// TwinCAT 3 PLC project MAXI
// ProgramVersion: 3.1.4024.0
// libraries:
//   Tc2_Standard, * (Beckhoff Automation GmbH)
//   Tc2_System, * (Beckhoff Automation GmbH)
//   Tc2_Utilities, * (Beckhoff Automation GmbH)
//   Tc3_Module, * (Beckhoff Automation GmbH)
// project tree:
//   DUTs/ BufferState.TcDUT
//   GVLs/ globals.TcGVL (not stored)
//   / PlcTask.TcTTO
//   POUs/ AnalogInput.TcPOU, FemtoCtrl.TcPOU, FilterRingBuffer.TcPOU (not stored), FlowMeter.TcPOU, LED.TcPOU, MAIN.TcPOU, ValueBuffer.TcPOU
// real-time tasks:
//   TASK PlcTask: cycle T#1ms, priority 20, ADS port 350
// I/O:
//   DEVICE Device 1 (EtherCAT), AmsNetId 5.82.117.74.2.1
//     Term 1 (EK1200) [EK1200-5000 EtherCAT Power supply (2A E-Bus)]
//       Term 2 (EL2595) [EL2595 1Ch. LED constant current terminal]
//       Term 3 (EL2595) [EL2595 1Ch. LED constant current terminal]
//       Term 4 (EL3102) [EL3102 2Ch. Ana. Input +/-10V, Diff.]
//       Term 5 (ELM3004-0000) [ELM3004-0000 4Ch. Ana. Input +/-30V, 24 bit, high precision]
//       Term 6 (EL9505) [EL9505 Power supply terminal 5V]
//       Term 7 (EL1124) [EL1124 4Ch. Dig. Input 5V, 10µs, Sensor Power]
//       Term 8 (EL2124) [EL2124 4Ch. Dig. Output 5V, 20mA]
//       Term 9 (EL2124) [EL2124 4Ch. Dig. Output 5V, 20mA]
//       Term 10 (EL2124) [EL2124 4Ch. Dig. Output 5V, 20mA]
//       Term 11 (EL9011) [EL9011 End Terminal]
// variable links:
//   MAXI/MAXI Instance <-> Device 1 (EtherCAT)/Term 1 (EK1200)/Term 2 (EL2595)
//     PlcTask Inputs/MAIN.LedBlue.bOutputActive <-> DOX Status/Status/Output active
//     PlcTask Inputs/MAIN.LedBlue.nCurrent <-> DOX Synchron info data/Info data 2
//     PlcTask Outputs/MAIN.LedBlue.bOutputSetpoint <-> DOX Control/Control/Output
//   MAXI/MAXI Instance <-> Device 1 (EtherCAT)/Term 1 (EK1200)/Term 3 (EL2595)
//     PlcTask Inputs/MAIN.LedWhite.bOutputActive <-> DOX Status/Status/Output active
//     PlcTask Inputs/MAIN.LedWhite.nCurrent <-> DOX Synchron info data/Info data 2
//     PlcTask Outputs/MAIN.LedWhite.bOutputSetpoint <-> DOX Control/Control/Output
//   MAXI/MAXI Instance <-> Device 1 (EtherCAT)/Term 1 (EK1200)/Term 5 (ELM3004-0000)
//     PlcTask Inputs/MAIN.ADC{1..4}.nRawValue <-> PAI Samples 1 Channel {1..4}/Samples[0]  (4 links)
//   MAXI/MAXI Instance <-> Device 1 (EtherCAT)/Term 1 (EK1200)/Term 7 (EL1124)
//     PlcTask Inputs/MAIN.Femto1.bOverload <-> Channel 1/Input
//     PlcTask Inputs/MAIN.Femto2.bOverload <-> Channel 3/Input
//     PlcTask Inputs/MAIN.flowmeter.bReedSwitch <-> Channel 2/Input
//   MAXI/MAXI Instance <-> Device 1 (EtherCAT)/Term 1 (EK1200)/Term 8 (EL2124)
//     PlcTask Outputs/MAIN.Femto1.bGainMode <-> Channel 4/Output
//     PlcTask Outputs/MAIN.Femto1.nGainBits <-> Channel 1/Output
//     PlcTask Outputs/MAIN.Femto1.nGainBits @bit 1 <-> Channel 2/Output
//     PlcTask Outputs/MAIN.Femto1.nGainBits @bit 2 <-> Channel 3/Output
//   MAXI/MAXI Instance <-> Device 1 (EtherCAT)/Term 1 (EK1200)/Term 9 (EL2124)
//     PlcTask Outputs/MAIN.Femto2.bGainMode <-> Channel 4/Output
//     PlcTask Outputs/MAIN.Femto2.nGainBits <-> Channel 1/Output
//     PlcTask Outputs/MAIN.Femto2.nGainBits @bit 1 <-> Channel 2/Output
//     PlcTask Outputs/MAIN.Femto2.nGainBits @bit 2 <-> Channel 3/Output

CONFIGURATION MAXI
    RESOURCE PLC ON TwinCAT3
        TASK PlcTask(INTERVAL := T#1ms, PRIORITY := 20);
        PROGRAM MAIN WITH PlcTask : MAIN;
    END_RESOURCE
END_CONFIGURATION

// ---- DUTs/BufferState.TcDUT
{attribute 'qualified_only'}
{attribute 'strict'}
TYPE BufferState :
(
	INIT, IDLE, STORING, FULL
);
END_TYPE

// ---- POUs/MAIN.TcPOU
PROGRAM MAIN
VAR
	LedBlue: LED;
	LedWhite: LED;
	Femto1: FemtoCtrl;
	Femto2: FemtoCtrl;
	ADC1: AnalogInput;
	ADC2: AnalogInput;
	ADC3: AnalogInput;
	ADC4: AnalogInput;
	bStartBuffer: BOOL := TRUE;
	bPrepareBuffer: BOOL := FALSE;
	nAdcBufferSize: UDINT := 1000; // size of array for dedicated acquisitions 
	bStopAdcBuffer: BOOL := FALSE;
	flowmeter: FlowMeter;
	sCommand: STRING := '';
	bCommandExecute: BOOL := FALSE;
	sCommandResult: STRING := '';
	fb_Shutdown: NT_Shutdown;
END_VAR

LedBlue();
LedWhite();
ADC1();
ADC2();
ADC3();
ADC4();

flowmeter();

IF bPrepareBuffer THEN
	nAdcBufferSize := ADC1.valuebuffer.PrepareBuffer(nNumValues:=nAdcBufferSize);
	nAdcBufferSize := ADC2.valuebuffer.PrepareBuffer(nNumValues:=nAdcBufferSize);
	nAdcBufferSize := ADC3.valuebuffer.PrepareBuffer(nNumValues:=nAdcBufferSize);
	nAdcBufferSize := ADC4.valuebuffer.PrepareBuffer(nNumValues:=nAdcBufferSize);
	bPrepareBuffer := FALSE;
END_IF

IF bStopAdcBuffer THEN
	ADC1.valuebuffer.StopBuffer();
	ADC2.valuebuffer.StopBuffer();
	ADC3.valuebuffer.StopBuffer();
	ADC4.valuebuffer.StopBuffer();
	bStopAdcBuffer := FALSE;
END_IF

IF bStartBuffer THEN
	ADC1.valuebuffer.StartBuffer();
	ADC2.valuebuffer.StartBuffer();
	ADC3.valuebuffer.StartBuffer();
	ADC4.valuebuffer.StartBuffer();
	bStartBuffer := FALSE;
END_IF

IF bCommandExecute THEN
	IF sCommand = 'SHUTDOWN' THEN
		fb_Shutdown(NETID:='', DELAY:=0, START:=bCommandExecute);
		sCommandResult := 'shutting down';
	ELSE
		sCommandResult := 'unknown command';
	END_IF
	bCommandExecute := FALSE;
END_IF

END_PROGRAM

// ---- POUs/LED.TcPOU
FUNCTION_BLOCK LED
VAR
	bOutputActive AT %I*: BOOL;
	bOutputSetpoint AT %Q*: BOOL;
	nCurrent AT %I*: UINT;
	nOutputCurrent: UINT;
END_VAR

IF bOutputActive THEN
	nOutputCurrent := nCurrent;
ELSE
	nOutputCurrent := 0;
END_IF

END_FUNCTION_BLOCK

// ---- POUs/FemtoCtrl.TcPOU
FUNCTION_BLOCK FemtoCtrl
VAR
	nGainBits AT %Q*: WORD; // assign multiple output bits with correct offset
	bGainMode AT %Q*: BOOL := TRUE; // TRUE: low noise, FALSE: high speed
	bOverload AT %I*: BOOL;
END_VAR

METHOD GetGain : WORD
VAR_INPUT
END_VAR
GetGain := nGainBits;
END_METHOD

METHOD GetGainMode : BOOL
VAR_INPUT
END_VAR
GetGainMode := bGainMode;
END_METHOD

METHOD GetOverload : BOOL
VAR_INPUT
END_VAR
GetOverload := bOverload;
END_METHOD

METHOD SetGain
VAR_INPUT
	nGain: WORD;
END_VAR
nGainBits := nGain;
END_METHOD

METHOD SetGainMode
VAR_INPUT
	bGainHigh: BOOL;
END_VAR
bGainMode := bGainHigh;
END_METHOD

END_FUNCTION_BLOCK

// ---- POUs/AnalogInput.TcPOU
FUNCTION_BLOCK AnalogInput
VAR
	nMaxRawValue: REAL := 7812500;  // for 24 bit device, e.g. ELM300x - check manual
	nRawValue AT %I*: DINT; // signed 32 bit integer representing full value range
	fMaxVoltage: REAL := 10; // measurement range
	valuebuffer: ValueBuffer; // buffer for timed measurements
	filterbuffer: FilterRingBuffer;
	nFilterSize: UDINT := 100;
	fVoltage: REAL;
	fVoltageFiltered: REAL; // running average filter
END_VAR

fVoltage := fMaxVoltage * DINT_TO_REAL(nRawValue) / nMaxRawValue;  

IF filterbuffer.nBufferSize <> nFilterSize THEN
	nFilterSize := filterbuffer.SetFilterSize(nFilterSize);
END_IF
filterbuffer.Store(fVoltage);
fVoltageFiltered := filterbuffer.CalculateMean();

valuebuffer(fValue:=fVoltage);  // makes sure buffer in initialized and calls StoreValueConditional

END_FUNCTION_BLOCK

// ---- POUs/ValueBuffer.TcPOU
FUNCTION_BLOCK ValueBuffer
VAR_INPUT
	fValue : REAL;
END_VAR
VAR
	values: ARRAY[0 .. globals.MAX_BUFFER_LENGTH] OF REAL;
	bInitialized: BOOL:=FALSE;
	nStoreEveryNthValue : UINT:=1;
	nCurrentIndex : UDINT:=1;
	eBufState : BufferState:=BufferState.INIT;
	nBufSize : UDINT:=1000;
	nTickCount : UDINT;
END_VAR

IF NOT bInitialized THEN
	// removed: dynamic memory allocation
	// reason: couldn't find a way to read via pyads (Error 1793 "Service is not supported by server")
	bInitialized := TRUE;
	eBufState := BufferState.IDLE;
END_IF

StoreValueConditional(fValue);

METHOD PUBLIC PrepareBuffer
VAR_INPUT
	nNumValues: UDINT;
END_VAR
VAR_OUTPUT
	nNumPrepared: UDINT;
END_VAR
VAR
	n: UDINT;
END_VAR
IF eBufState = BufferState.IDLE OR eBufState = BufferState.FULL THEN
	// IF nNumValues <> nBufSize THEN
		// fbMemoryBuffer.Resize(nSize:=nNumValues * SIZEOF(REAL), bPreserve:=FALSE, bReset:=TRUE);
		// values := fbMemoryBuffer.pBuffer;
		// nBufSize := nNumValues;
	// ELSE
		// fbMemoryBuffer.Clear();
	// END_IF
	nBufSize := MIN(nNumValues, globals.MAX_BUFFER_LENGTH);
	nNumPrepared := nBufSize;
	FOR n := 0 TO nBufSize DO
		values[n] := 0;
	END_FOR
eBufState := BufferState.IDLE;
nCurrentIndex := 0;
nTickCount := 0;
END_IF
END_METHOD

METHOD StartBuffer
IF eBufState = BufferState.IDLE THEN
	eBufState := BufferState.STORING;
END_IF
END_METHOD

METHOD StopBuffer
eBufState := BufferState.FULL;
END_METHOD

METHOD StoreValueConditional // Store value in buffer if tick count MOD buffer rate equals 0 
VAR_INPUT
	fValue : REAL;
END_VAR
IF eBufState = BufferState.STORING THEN
	IF (nTickCount MOD nStoreEveryNthValue) = 0 THEN
		values[nCurrentIndex] := fValue;
		nCurrentIndex := nCurrentIndex + 1;
	END_IF
	nTickCount := nTickCount + 1;
END_IF

IF nCurrentIndex >= nBufSize OR nCurrentIndex >= globals.MAX_BUFFER_LENGTH THEN
	eBufState := BufferState.FULL;
END_IF
END_METHOD

END_FUNCTION_BLOCK

// ---- POUs/FlowMeter.TcPOU
FUNCTION_BLOCK FlowMeter
VAR CONSTANT
	MAXLEN: UINT := 1000;
	TIMEUNITSPERSECOND: LINT := 10_000_000; // 100 ns per step
END_VAR
VAR
	fFrequencyToFlowScale: REAL := 0.28;
	fFlowRate: REAL;
	bReedSwitch AT %I*: BOOL;
	nIndex: UINT;
	timestamps: ARRAY [0..MAXLEN] OF ULINT;
	nTimeNow: ULINT; // 100 ns per unit
	nTriggerCount: UINT;
	nLoopIndex: UINT;
	trigger: R_TRIG;
END_VAR

// Koolance INS-FM19 flow meter
// simple reed contact switch
// frequency directly proportional to flow rate
// typical frequencies are <30 Hz, so no fast counter required

nTimeNow := F_GetSystemTime();
trigger(CLK:=bReedSwitch);
IF trigger.Q THEN
	timestamps[nIndex] := nTimeNow;
	nIndex := (nIndex + 1) MOD  MAXLEN;
END_IF

nTriggerCount := 0;
FOR nLoopIndex := 0 TO MAXLEN DO
	IF (ULINT_TO_LINT(nTimeNow) - ULINT_TO_LINT(timestamps[nLoopIndex])) < TIMEUNITSPERSECOND THEN
		nTriggerCount := nTriggerCount + 1;
	END_IF
END_FOR

fFlowRate := fFrequencyToFlowScale * nTriggerCount;

END_FUNCTION_BLOCK
